// TIA Portal V20 export
VAR_GLOBAL   // PLC tag table "EVT_Const_Gen"
END_VAR
VAR_GLOBAL CONSTANT   // user constants
   EVT_CAPACITY : Int := 1000;   // EVTLOG entries / EVTLOG 항목 수
   EVT_LAST : Int := 999;   // EVTLOG.Entry upper bound / EVTLOG.Entry 상한
   EVT_MIN_LEVEL_DEFAULT : USInt := 2;   // Default Cfg.MinLevel / Cfg.MinLevel 기본값
   EVT_MAX_PER_SCAN_DEFAULT : Int := 32;   // Default Cfg.MaxPerScan / Cfg.MaxPerScan 기본값
   EVT_CATMASK_ALL : DWord := 16#0003FFFE;   // Cfg.CatMask, every category / Cfg.CatMask 전 분류
   EVT_LVL_TRACE : USInt := 0;   // Level TRACE / 레벨 TRACE
   EVT_LVL_DEBUG : USInt := 1;   // Level DEBUG / 레벨 DEBUG
   EVT_LVL_INFO : USInt := 2;   // Level INFO / 레벨 INFO
   EVT_LVL_WARN : USInt := 3;   // Level WARN / 레벨 WARN
   EVT_LVL_ERROR : USInt := 4;   // Level ERROR / 레벨 ERROR
   EVT_CAT_SYS : USInt := 1;   // Category SYS (CatMask bit 1) / 분류 SYS
   EVT_CAT_MODE : USInt := 2;   // Category MODE (CatMask bit 2) / 분류 MODE
   EVT_CAT_STEP : USInt := 3;   // Category STEP (CatMask bit 3) / 분류 STEP
   EVT_CAT_TASK : USInt := 4;   // Category TASK (CatMask bit 4) / 분류 TASK
   EVT_CAT_CMD : USInt := 5;   // Category CMD (CatMask bit 5) / 분류 CMD
   EVT_CAT_ALARM : USInt := 6;   // Category ALARM (CatMask bit 6) / 분류 ALARM
   EVT_CAT_GRIP : USInt := 7;   // Category GRIP (CatMask bit 7) / 분류 GRIP
   EVT_CAT_DRIVE : USInt := 8;   // Category DRIVE (CatMask bit 8) / 분류 DRIVE
   EVT_CAT_SAFETY : USInt := 9;   // Category SAFETY (CatMask bit 9) / 분류 SAFETY
   EVT_CAT_SENSOR : USInt := 10;   // Category SENSOR (CatMask bit 10) / 분류 SENSOR
   EVT_CAT_MEAS : USInt := 11;   // Category MEAS (CatMask bit 11) / 분류 MEAS
   EVT_CAT_ILOCK : USInt := 12;   // Category ILOCK (CatMask bit 12) / 분류 ILOCK
   EVT_CAT_ANTICOL : USInt := 13;   // Category ANTICOL (CatMask bit 13) / 분류 ANTICOL
   EVT_CAT_COMM : USInt := 14;   // Category COMM (CatMask bit 14) / 분류 COMM
   EVT_CAT_DATA : USInt := 15;   // Category DATA (CatMask bit 15) / 분류 DATA
   EVT_CAT_STATION : USInt := 16;   // Category STATION (CatMask bit 16) / 분류 STATION
   EVT_CAT_SCEN : USInt := 17;   // Category SCEN (CatMask bit 17) / 분류 SCEN
   EVT_SYS_STARTUP : UInt := 101;   // SYS INFO / PLC 기동 {a:bits:startup}
   EVT_SYS_PROG_ERROR : UInt := 102;   // SYS ERROR / Programming error : block {src}, Fault_ID {a:hex}, DB {b}
   EVT_SYS_CYCLE_OVERRUN : UInt := 103;   // SYS ERROR / Cycle time error : Fault_ID {a:hex}
   EVT_SYS_CLOCK_SET : UInt := 104;   // SYS WARN / 시계 보정 {a} ms
   EVT_SYS_LOGGER_DROP : UInt := 105;   // SYS WARN / 로거 누락 : Dropped {a} (MaxPerScan 초과)
   EVT_SYS_LOGGER_SLOW : UInt := 106;   // SYS WARN / 로거 실행 시간 MaxRunUs {a} µs
   EVT_SYS_IP_CONFIG : UInt := 107;   // SYS INFO / IP 설정 {src:ip_if} {b:ip_result} (STATUS {a:hex})
   EVT_SYS_GCS_TIME_STALE : UInt := 108;   // SYS WARN / GCS NTP 갱신 {b:stall} ({a} ms)
   EVT_MODE_CHANGED : UInt := 201;   // MODE INFO / {b:mode} → {a:mode}
   EVT_MODE_REJECTED : UInt := 202;   // MODE WARN / 모드 요청 거부 {b:mode} → {a:mode}
   EVT_MODE_FAULT_RESET : UInt := 206;   // MODE INFO / Fault reset {a:reset_result} (FaultCode[0] {b})
   EVT_MODE_OPTION : UInt := 207;   // MODE WARN / Option {src:option} {a:onoff}
   EVT_MODE_GRM_OPTION : UInt := 212;   // MODE WARN / Option {src:grm_option} {a:onoff}
   EVT_MODE_GRM_FORCE : UInt := 213;   // MODE WARN / {src:grm_force} {a:onoff}
   EVT_CMD_GCS_NEW : UInt := 520;   // CMD INFO / GR{src} 새 명령 {b:cmd_type} · Cell {a}
   EVT_CMD_GCS_ACK : UInt := 521;   // CMD INFO / GR{src} 명령 ack {b:cmd_type} ({a} ms)
   EVT_CMD_GCS_OVERWRITE : UInt := 522;   // CMD WARN / GR{src} ack 전 덮어씀 : 이전 {b:cmd_type} WorkId {a}
   EVT_CMD_GCS_BITS : UInt := 523;   // CMD INFO / GR{src} 명령 비트 {a:bits:gcs_cmd_bits} (이전 {b:bits:gcs_cmd_bits})
   EVT_CMD_GCS_PARTIAL : UInt := 524;   // CMD WARN / GR{src} 헤더 일부만 씀 (CMDRetry) {b:cmd_type}
   EVT_CMD_GCS_RESEND : UInt := 525;   // CMD WARN / GR{src} 30 s 무응답 재전송 {b:cmd_type} SEQ {a}
   EVT_CMD_GCS_ACCEPT_HOLD : UInt := 526;   // CMD DEBUG / GR{src} Accept 보류 {a:onoff}
   EVT_ALM_RAISED : UInt := 601;   // ALARM ERROR / {alarm} 발생 (step {b})
   EVT_ALM_CLEARED : UInt := 602;   // ALARM INFO / {alarm} 해제
   EVT_ALM_RESET : UInt := 603;   // ALARM INFO / {src:alarm_area} reset ({a} bits set)
   EVT_ALM_TO_FAULT : UInt := 604;   // ALARM ERROR / FAULT 전환 : 첫 코드 {a}
   EVT_SAFE_EMS : UInt := 901;   // SAFETY ERROR / EMS {a:onoff}
   EVT_SAFE_IO_FORCE : UInt := 903;   // SAFETY WARN / {src:io_force} {a:onoff}
   EVT_SAFE_GRM_EMS : UInt := 905;   // SAFETY ERROR / {src:ems_src} {a:onoff}
   EVT_SAFE_ZONE : UInt := 906;   // SAFETY WARN / Area{src} {a:bits:zone_bits} (이전 {b:bits:zone_bits})
   EVT_SAFE_DOOR : UInt := 907;   // SAFETY INFO / Door {src} {b:door_status} → {a:door_status}
   EVT_SAFE_DOOR_ERROR : UInt := 908;   // SAFETY ERROR / GR{src} 요청 없이 도어 열림 {a:onoff}
   EVT_SAFE_HMI_BLOCK : UInt := 909;   // SAFETY WARN / HMI 조작 차단 {a:onoff}
   EVT_SAFE_COMMISSION_WIPE : UInt := 910;   // SAFETY WARN / SafetyCommission : PARA ZoneNo/ioModuleNo {a} 개 지움
   EVT_SAFE_GRM_INPUT : UInt := 911;   // SAFETY WARN / {src:grm_input} {a:onoff}
   EVT_SAFE_GRM_BUTTON : UInt := 912;   // SAFETY DEBUG / {src:grm_button} {a:onoff}
   EVT_SNS_MODULE_DIAG : UInt := 1004;   // SENSOR WARN / Module diag {src:module_diag} : {a:bits:diag_bits}
   EVT_SNS_PORT_LINK : UInt := 1006;   // SENSOR WARN / PN module {src} (module*10+port) {b:port_link} → {a:port_link}
   EVT_COM_LINK : UInt := 1401;   // COMM WARN / {src:peer} link {a:onoff} (끊김 {b} ms)
   EVT_COM_BLOCK_ERR : UInt := 1402;   // COMM WARN / {src:comm_block} error STATUS {a:hex}
   EVT_COM_HEARTBEAT : UInt := 1404;   // COMM WARN / {src:peer} heartbeat {b:stall} ({a} ms)
   EVT_COM_GET_FAIL : UInt := 1407;   // COMM DEBUG / GET NDR 없음 STATUS {a:hex}
   EVT_COM_BSEND_DONE : UInt := 1408;   // COMM INFO / GR{src} BSEND 완료 {b:cmd_type} {a:bits:gcs_cmd_bits}
   EVT_COM_RECV_GAP : UInt := 1409;   // COMM WARN / GR{src} BRCV 간격 {a} ms
   EVT_COM_GR_CMD_ERROR : UInt := 1410;   // COMM WARN / GR{src} 명령 오류 StatusCode {a}.{b}
   EVT_COM_GRM_TO_GR : UInt := 1411;   // COMM INFO / GRM→GR{src} {a:bits:grm_send_status} (이전 {b:bits:grm_send_status})
   EVT_COM_HMI_PANEL : UInt := 1412;   // COMM WARN / HMI 판넬 (MTP) heartbeat {b:stall} ({a} ms)
   EVT_COM_GRM_BLOCK_ERR : UInt := 1413;   // COMM WARN / GR{src} {b:comm_block} error STATUS {a:hex}
   EVT_DATA_CSV : UInt := 1501;   // DATA INFO / CSV {src:csv_kind} : {a:csv_result} (STATUS {b:hex})
   EVT_DATA_PARA_SECTION : UInt := 1508;   // DATA INFO / PARA.{src:para_section} 변경 (checksum {b:hex} → {a:hex})
   EVT_DATA_GRM_PARA_SECTION : UInt := 1510;   // DATA INFO / PARA.{src:grm_para_section} 변경 (checksum {b:hex} → {a:hex})
   EVT_DATA_CSV_ROW : UInt := 1511;   // DATA WARN / CSV {src:csv_kind} 잘못된 행 {a} ({b:csv_dir})
   EVT_ST_MEAS_COMP : UInt := 1601;   // STATION INFO / St{src} GCS MeasComp {a:onoff}
   EVT_ST_TRACK_CLEAR : UInt := 1602;   // STATION INFO / St{src} GCS 트래킹 명령 : {a:track_clear} ({b})
   EVT_ST_CV_IN : UInt := 1603;   // STATION INFO / St{src} CV→GRM {a:bits:pi_bits} (이전 {b:bits:pi_bits})
   EVT_ST_CV_OUT : UInt := 1604;   // STATION INFO / St{src} GRM→CV {a:bits:cv_out} (이전 {b:bits:cv_out})
   EVT_ST_CVNO_REASON : UInt := 1605;   // STATION INFO / St{src} CVNO 이유 {a:bits:cvno_reason} (이전 {b:bits:cvno_reason})
   EVT_ST_MEAS : UInt := 1606;   // STATION INFO / St{src} 측정 {a:st_meas} OD {b/10} mm
   EVT_ST_MEAS_OFFSET : UInt := 1607;   // STATION INFO / St{src} 측정 TaskOffset X {a/10} · Y {b/10} mm
   EVT_ST_STATUS : UInt := 1608;   // STATION WARN / St{src} {a:bits:st_status} (이전 {b:bits:st_status})
   EVT_ST_TRACKING : UInt := 1609;   // STATION INFO / St{src} 트래킹 {a:track_cause} ({b})
   EVT_ST_HMI_OP : UInt := 1610;   // STATION INFO / St{src} {a:st_hmi_op}
   EVT_ST_ROBOT_OVER : UInt := 1611;   // STATION DEBUG / St{src} GR{a} 위 {b:onoff}
   EVT_SC_RUN : UInt := 1701;   // SCEN INFO / GR{src} 시나리오 {a:onoff} (List {b})
   EVT_SC_TASK : UInt := 1702;   // SCEN INFO / GR{src} 시나리오 작업 {a:sc_task} (index {b})
   EVT_SC_BLOCKED : UInt := 1703;   // SCEN WARN / GR{src} 시나리오 전송 보류 {a:bits:sc_block} (index {b})
   EVT_TEACH_RUN : UInt := 1704;   // SCEN INFO / GR{src} Teach {a:onoff} (index {b})
   EVT_TEACH_TASK : UInt := 1705;   // SCEN INFO / GR{src} Teach 이동 {a:teach_task} (Cell index {b})
   EVT_TEACH_CELL_Z : UInt := 1706;   // SCEN WARN / Cell {src} Z {b/10} → {a/10} mm (바닥 측정)
   EVT_CELL_EDIT : UInt := 1707;   // SCEN INFO / Cell {src} {a:cell_edit} (CELL.Count {b})
   EVT_ALARM_AREA_FAULT : UInt := 1;   // alarm_area = FAULT
   EVT_ALARM_AREA_WARN : UInt := 2;   // alarm_area = WARN
   EVT_ALARM_AREA_EVENT : UInt := 3;   // alarm_area = EVENT
   EVT_ALARM_AREA_TASK : UInt := 4;   // alarm_area = TASK
   EVT_AUTO_STOP_PB_STOP : UInt := 1;   // auto_stop = PB_Stop
   EVT_AUTO_STOP_ALLSTOP : UInt := 2;   // auto_stop = AllStop
   EVT_AUTO_STOP_EMS : UInt := 3;   // auto_stop = EMS
   EVT_AUTO_STOP_SSW_AUTO_OFF : UInt := 4;   // auto_stop = SSW_Auto off
   EVT_CANCEL_RESULT_OK : UInt := 1;   // cancel_result = OK
   EVT_CANCEL_RESULT_REFUSED_F6020 : UInt := 2;   // cancel_result = Refused (F6020)
   EVT_CELL_EDIT_APPLY : UInt := 1;   // cell_edit = Apply
   EVT_CELL_EDIT_SAVE : UInt := 2;   // cell_edit = Save
   EVT_CELL_EDIT_ADD : UInt := 3;   // cell_edit = Add
   EVT_CELL_EDIT_CREATE : UInt := 4;   // cell_edit = Create
   EVT_CELL_EDIT_DELETE : UInt := 5;   // cell_edit = Delete
   EVT_CELL_EDIT_CSV_IMPORT : UInt := 6;   // cell_edit = CSV import
   EVT_CMD_SRC_OPC : UInt := 1;   // cmd_src = OPC
   EVT_CMD_SRC_HMI : UInt := 2;   // cmd_src = HMI
   EVT_CMD_SRC_HMI_FORCE : UInt := 3;   // cmd_src = HMI Force
   EVT_CMD_SRC_SOCKET : UInt := 4;   // cmd_src = Socket
   EVT_COMM_BLOCK_BSEND : UInt := 1;   // comm_block = BSEND
   EVT_COMM_BLOCK_BRCV : UInt := 2;   // comm_block = BRCV
   EVT_COMM_BLOCK_GET : UInt := 3;   // comm_block = GET
   EVT_CSV_RESULT_IMPORT_REQUEST : UInt := 1;   // csv_result = Import request
   EVT_CSV_RESULT_IMPORT_DONE : UInt := 2;   // csv_result = Import done
   EVT_CSV_RESULT_IMPORT_TIMEOUT : UInt := 3;   // csv_result = Import timeout
   EVT_CSV_RESULT_FILE_MISSING_DEFAULTS : UInt := 4;   // csv_result = File missing -> defaults
   EVT_CSV_RESULT_IMPORT_ERROR_TREATED_AS_DONE : UInt := 5;   // csv_result = Import error (treated as done)
   EVT_CSV_RESULT_EXPORT : UInt := 6;   // csv_result = Export
   EVT_CSV_RESULT_EXPORT_ERROR : UInt := 7;   // csv_result = Export error
   EVT_IP_IF_X1 : UInt := 1;   // ip_if = X1
   EVT_IP_IF_X2 : UInt := 2;   // ip_if = X2
   EVT_LEARN_PHASE_ACCEPTED : UInt := 1;   // learn_phase = Accepted
   EVT_LEARN_PHASE_DONE : UInt := 2;   // learn_phase = Done
   EVT_LEARN_PHASE_ERROR : UInt := 3;   // learn_phase = Error
   EVT_MANUAL_COMPLETE_REQUESTED : UInt := 1;   // manual_complete = Requested
   EVT_MANUAL_COMPLETE_REFUSED_AUTO_W6026 : UInt := 2;   // manual_complete = Refused AUTO (W6026)
   EVT_MANUAL_COMPLETE_GRIP_NG_F6022 : UInt := 3;   // manual_complete = Grip NG (F6022)
   EVT_MANUAL_COMPLETE_NO_ITEM_F6018 : UInt := 4;   // manual_complete = No item (F6018)
   EVT_MANUAL_COMPLETE_PENDING_CV_HANDOVER : UInt := 5;   // manual_complete = Pending CV handover
   EVT_MANUAL_COMPLETE_DONE : UInt := 6;   // manual_complete = Done
   EVT_PARA_SENSOR_GIDL_ZOFFSET : UInt := 1;   // para = Sensor.GIDL_ZOffset
   EVT_PARA_SENSOR_GIDF_ZOFFSET : UInt := 2;   // para = Sensor.GIDF_ZOffset
   EVT_PARA_SENSOR_GIDR_ZOFFSET : UInt := 3;   // para = Sensor.GIDR_ZOffset
   EVT_PARA_SENSOR_GIDB_ZOFFSET : UInt := 4;   // para = Sensor.GIDB_ZOffset
   EVT_PARA_DRIVE_HOMEPOS_X : UInt := 11;   // para = Drive.HomePos[X]
   EVT_PARA_DRIVE_HOMEPOS_Y : UInt := 12;   // para = Drive.HomePos[Y]
   EVT_PARA_DRIVE_HOMEPOS_Z : UInt := 13;   // para = Drive.HomePos[Z]
   EVT_PARA_DRIVE_HOMEPOS_G : UInt := 14;   // para = Drive.HomePos[G]
   EVT_PARA_DRIVE_RANGEMIN_X : UInt := 21;   // para = Drive.RangeMin[X]
   EVT_PARA_DRIVE_RANGEMIN_Y : UInt := 22;   // para = Drive.RangeMin[Y]
   EVT_PARA_DRIVE_RANGEMIN_Z : UInt := 23;   // para = Drive.RangeMin[Z]
   EVT_PARA_DRIVE_RANGEMIN_G : UInt := 24;   // para = Drive.RangeMin[G]
   EVT_PARA_DRIVE_RANGEMAX_X : UInt := 31;   // para = Drive.RangeMax[X]
   EVT_PARA_DRIVE_RANGEMAX_Y : UInt := 32;   // para = Drive.RangeMax[Y]
   EVT_PARA_DRIVE_RANGEMAX_Z : UInt := 33;   // para = Drive.RangeMax[Z]
   EVT_PARA_DRIVE_RANGEMAX_G : UInt := 34;   // para = Drive.RangeMax[G]
   EVT_PARA_DRIVE_MCS_TO_ACS_Z_0 : UInt := 41;   // para = Drive.MCS_TO_ACS[Z,0]
   EVT_PARA_DRIVE_MCS_TO_ACS_Z_1 : UInt := 42;   // para = Drive.MCS_TO_ACS[Z,1]
   EVT_PARA_DRIVE_MCS_TO_ACS_Z_2 : UInt := 43;   // para = Drive.MCS_TO_ACS[Z,2]
   EVT_PARA_DRIVE_ACS_TO_MCS_Z_0 : UInt := 44;   // para = Drive.ACS_TO_MCS[Z,0]
   EVT_PARA_DRIVE_ACS_TO_MCS_Z_1 : UInt := 45;   // para = Drive.ACS_TO_MCS[Z,1]
   EVT_PARA_DRIVE_ACS_TO_MCS_Z_2 : UInt := 46;   // para = Drive.ACS_TO_MCS[Z,2]
   EVT_PARA_MACHINE_XLENGTHFRONT : UInt := 51;   // para = Machine.XLengthFront
   EVT_PARA_MACHINE_XLENGTHREAR : UInt := 52;   // para = Machine.XLengthRear
   EVT_PARA_SENSOR_XACF_OFFSET : UInt := 53;   // para = Sensor.XACF_Offset
   EVT_PARA_SENSOR_XACR_OFFSET : UInt := 54;   // para = Sensor.XACR_Offset
   EVT_PARA_SENSOR_FLD_OFFSET : UInt := 55;   // para = Sensor.FLD_Offset
   EVT_PARA_MACHINE_G_OFFSET : UInt := 56;   // para = Machine.G_Offset
   EVT_PENDING_END_CV_HANDOVER : UInt := 1;   // pending_end = CV handover
   EVT_PENDING_END_AUTO_FORCED_W6024 : UInt := 2;   // pending_end = AUTO forced (W6024)
   EVT_PENDING_END_TIMEOUT_W6024 : UInt := 3;   // pending_end = Timeout (W6024)
   EVT_PENDING_END_DROPPED : UInt := 4;   // pending_end = Dropped
   EVT_PROC_TASK : UInt := 20;   // proc = Task
   EVT_PROC_INIT : UInt := 100;   // proc = Init
   EVT_PROC_CHANGEIP : UInt := 110;   // proc = ChangeIP
   EVT_PROC_HOMINGX : UInt := 121;   // proc = HomingX
   EVT_PROC_HOMINGY : UInt := 122;   // proc = HomingY
   EVT_PROC_HOMINGZ : UInt := 123;   // proc = HomingZ
   EVT_PROC_HOMINGG : UInt := 124;   // proc = HomingG
   EVT_PROC_INITPOS : UInt := 130;   // proc = InitPos
   EVT_PROC_MEASUREITEM : UInt := 140;   // proc = MeasureItem
   EVT_PROC_MANUALMEASURE : UInt := 141;   // proc = ManualMeasure
   EVT_PROC_CALIBRATIONZ : UInt := 150;   // proc = CalibrationZ
   EVT_PROC_CELLORIGINX : UInt := 161;   // proc = CellOriginX
   EVT_PROC_CELLORIGINY : UInt := 162;   // proc = CellOriginY
   EVT_RESET_RESULT_TRY : UInt := 1;   // reset_result = Try
   EVT_RESET_RESULT_OK : UInt := 2;   // reset_result = OK
   EVT_RESET_RESULT_FAIL : UInt := 3;   // reset_result = Fail
   EVT_SC_TASK_SENT : UInt := 1;   // sc_task = Sent
   EVT_SC_TASK_ACK : UInt := 2;   // sc_task = Ack
   EVT_SC_TASK_ACK_TIMEOUT : UInt := 3;   // sc_task = Ack timeout
   EVT_SC_TASK_WRAP_END : UInt := 4;   // sc_task = Wrap end
   EVT_ST_HMI_OP_FORCECOMPLETE : UInt := 1;   // st_hmi_op = ForceComplete
   EVT_ST_HMI_OP_SENSORAPPLY : UInt := 2;   // st_hmi_op = SensorApply
   EVT_ST_HMI_OP_SAVE : UInt := 3;   // st_hmi_op = Save
   EVT_ST_HMI_OP_TRACKINGERRORRESET : UInt := 4;   // st_hmi_op = TrackingErrorReset
   EVT_ST_MEAS_START : UInt := 1;   // st_meas = Start
   EVT_ST_MEAS_DONE : UInt := 2;   // st_meas = Done
   EVT_ST_MEAS_ERROR : UInt := 3;   // st_meas = Error
   EVT_ST_MEAS_DUPLICATE : UInt := 4;   // st_meas = Duplicate
   EVT_ST_MEAS_ERROR_X_OFFSET : UInt := 5;   // st_meas = Error X offset
   EVT_ST_MEAS_ERROR_Y_OFFSET : UInt := 6;   // st_meas = Error Y offset
   EVT_ST_MEAS_ERROR_DIAMETER : UInt := 7;   // st_meas = Error diameter
   EVT_ST_MEAS_NO_DATA_5_S : UInt := 8;   // st_meas = No data 5 s
   EVT_START_BLOCK_ROBOTUSE : UInt := 0;   // start_block = RobotUse
   EVT_START_BLOCK_POWERONDRIVE : UInt := 1;   // start_block = PowerOnDrive
   EVT_START_BLOCK_DRIVESYNC : UInt := 2;   // start_block = DriveSync
   EVT_START_BLOCK_GRM_CONNECTED : UInt := 3;   // start_block = GRM_Connected
   EVT_START_SRC_PB_START : UInt := 1;   // start_src = PB_Start
   EVT_START_SRC_GCS_COMMON_START : UInt := 2;   // start_src = GCS Common.Start
   EVT_TEACH_TASK_SENT : UInt := 1;   // teach_task = Sent
   EVT_TEACH_TASK_ACK : UInt := 2;   // teach_task = Ack
   EVT_TEACH_TASK_ACK_TIMEOUT : UInt := 3;   // teach_task = Ack timeout
   EVT_TEACH_TASK_NULL_CELL_STOP : UInt := 4;   // teach_task = Null cell stop
   EVT_TRACK_CAUSE_MEASURED : UInt := 1;   // track_cause = Measured
   EVT_TRACK_CAUSE_MOVED : UInt := 2;   // track_cause = Moved
   EVT_TRACK_CAUSE_ROBOT_PICK : UInt := 3;   // track_cause = Robot pick
   EVT_TRACK_CAUSE_GCS_CLEAR : UInt := 4;   // track_cause = GCS clear
   EVT_TRACK_CAUSE_HMI_CLEAR : UInt := 5;   // track_cause = HMI clear
   EVT_TRACK_CAUSE_HMI_SAVE : UInt := 6;   // track_cause = HMI save
   EVT_TRACK_CLEAR_ACCEPTED : UInt := 1;   // track_clear = Accepted
   EVT_TRACK_CLEAR_REJECTED_ITEM_DETECTED : UInt := 2;   // track_clear = Rejected item detected
   EVT_TRACK_CLEAR_UNSUPPORTED_CMD : UInt := 3;   // track_clear = Unsupported cmd
   EVT_UNUSED_CMD_STOP_FAST : UInt := 1;   // unused_cmd = Stop.Fast
   EVT_UNUSED_CMD_STOP_CYCLE : UInt := 2;   // unused_cmd = Stop.Cycle
   EVT_UNUSED_CMD_COMMON_INITIALIZING : UInt := 3;   // unused_cmd = Common.Initializing
   EVT_UNUSED_CMD_JOG : UInt := 4;   // unused_cmd = Jog
   EVT_UNUSED_CMD_HOME : UInt := 5;   // unused_cmd = Home
   EVT_UNUSED_CMD_MAINTPOS : UInt := 6;   // unused_cmd = MaintPos
   EVT_UNUSED_CMD_CELLORIGIN : UInt := 7;   // unused_cmd = CellOrigin
   EVT_UNUSED_CMD_CHANGEMODE : UInt := 8;   // unused_cmd = ChangeMode
END_VAR
